FUNCTION_BLOCK ASR2_4EVENTS_TO_SR2 (* Composite FB for convert 4 EVENTS to ASR2 *)
  (* Standard: 61499-2; Description: Copyright (c) 2024 HR Agrartechnik GmbH This program and the accompanying materials are made available under the terms of the Eclipse Public License 2.0 which is available at https://www.eclipse.org/legal/epl-2.0/ SPDX-License-Identifier: EPL-2.0 *)
  (* Version 1.0, 2024-04-24, Franz Höpfinger, HR Agrartechnik GmbH *)
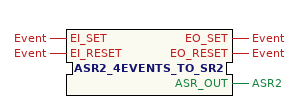
  EVENT_INPUT
    EI_SET; (* Set / Switch on *)
    EI_RESET; (* Reset / Switch off *)
  END_EVENT
  EVENT_OUTPUT
    EO_SET; (* Set / Switch on *)
    EO_RESET; (* Reset / Switch off *)
  END_EVENT
  PLUGS
    ASR_OUT : ASR2; (* Adapter Output *)
  END_PLUGS
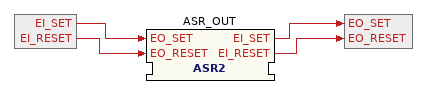
  EVENT_CONNECTIONS
    ASR_OUT.EI_SET TO EO_SET;
    ASR_OUT.EI_RESET TO EO_RESET;
    EI_SET TO ASR_OUT.EO_SET;
    EI_RESET TO ASR_OUT.EO_RESET;
  END_CONNECTIONS
END_FUNCTION_BLOCK
